Staubli VAL3: userPage7En.dtx

public num nBottomX[2]
  [0] = 21
  [1] = 21
public num nBottomY = 10
num nFirst
num nKey = 255
num nOldValue[2]
  [0] = 200
  [1] = 200
public num nPage = 100000
public num nTopX[2]
  [0] = 17
  [1] = 17
public num nTopY
public num nView
string sExample1
string sExample2
public string sItems[17]
  [0] = "Name: > "
  [1] = "coord  X > 680.52"
  [2] = "coord  Y > -61.92"
  [3] = "coord  Z > 300.32"
  [4] = "coord RX > -10   "
  [5] = "coord RY > 175.5 "
  [6] = "coord RZ > 68.47"
  [7] = "Axis pos > 90   "
  [8] = "MoveType > Linear"
  [9] = "Speed    > 600 mm/s"
  [10] = "Accelerat> 200 %"
  [11] = "Stop  > [ ]"
  [12] = "Blend[x] > 30 mm"
  [13] = "Action : 1> "
  [14] = "Action : 2> "
  [15] = "Action : 3> "
  [16] = "Anticipation > 0 mm"
string sMenu
string sMessage[3]
  [0] = "Insert the speed, all the points that"
  [1] = "have the same speeed will be change,"
  [2] = "use mm/sec >600"
string sTab[4]
  [0] = "test1"
  [1] = "test2"
  [2] = "test3"
  [3] = "test4"
string sTitle
bool Show
bool bReadWrite[17]
  [0] = true
  [1] = true
  [2] = true
  [3] = true
  [4] = true
  [5] = true
  [6] = true
  [7] = true
  [8] = true
  [9] = true
  [10] = true
  [11] = true
  [12] = true
  [13] = true
  [14] = true
  [15] = true
  [16] = true
public bool bShowDialog
public bool bUseEscape = true
public bool bUseRefresh
screen scr
